(* IEC 61131-3 sources: cds-text-sync-reference-project/project-view/PLC/PLC Logic/ST_Application/02_Object_GVL, 3 files *)

(* ---- _01_GVL.st ---- *)
{attribute 'qualified_only'}
VAR_GLOBAL
END_VAR
VAR_GLOBAL
	xSysRestart : BOOL;         // Global system restart command
	rMainPressure : _03_DUT_Alias; // Using Alias type (renamed to match object)
	stActivePump : _01_DUT_STRUCTURE; // Using Structure type (renamed to match object)
	eCurrentState : _02_DUT_Enumeration; // Using Enum type (renamed to match object)
	uStatus : _04_DUT_UNION; // Using Union type (renamed to match object)
END_VAR

VAR_GLOBAL CONSTANT
	MAX_PUMPS : INT := 4;
	PI : REAL := 3.141592;
END_VAR

VAR_GLOBAL RETAIN
	diTotalCycleCounter : DINT; // Non-volatile counter
END_VAR

(* ---- _02_TaskLocalGVL.st ---- *)
(* cds-text-sync: TypeGuid="{c2cda7a9-0ba4-4146-b563-22a42fa0eb72}" *)
// [INFO] Task with write access: Task (set manually in CODESYS, not restored by import)
{attribute 'qualified_only'}
VAR_GLOBAL
	iInteger : INT; // [INFO] Integer variable
END_VAR

(* ---- _03_NVL_sender.st ---- *)
{attribute 'qualified_only'}
VAR_GLOBAL
	someInteger : INT; //Integer value
END_VAR
